// TwinCAT 3 PLC project mdx91test
// ProgramVersion: 3.1.4023.0
// libraries:
//   Tc2_Standard, * (Beckhoff Automation GmbH)
//   Tc2_System, * (Beckhoff Automation GmbH)
//   Tc3_Module, * (Beckhoff Automation GmbH)
// project tree:
//   / PlcTask.TcTTO
//   POUs/ MAIN.TcPOU
//   POUs/SEW_MOVIKITpositioningDrive/ FB_MOVIKITpositioningDrive.TcPOU
//   POUs/SEW_MOVIKITpositioningDrive/General/ eMOVIKITpositioningDrive_ApplMode.TcDUT, stMOVIKITpositioningDrive.TcDUT, stPositioning_IN.TcDUT, stPositioning_OUT.TcDUT
// real-time tasks:
//   TASK PlcTask: cycle T#10ms, priority 20, ADS port 350
// motion (NC):
//   TASK NC-Task 1 SAF: cycle T#2ms, priority 4, ADS port 501
//   TASK NC-Task 1 SVB: cycle T#10ms, priority 8, ADS port 511
//   AXIS Axis 1 (id 1)
//     OtherSettings: AllowMotionCmdToSlave=true
//     encoder EncType=1
//     drive DrvType=5
//       Analog: TorqueSetpointScale=10, ScaleFactorActTorque=0.1
//       TimeComp: TaskDelayCycles=1
//     controller CtrType=1
//       CtrPara: PriorControlFactor=1
//         Observer: BandWidth=20
// I/O:
//   DEVICE Device 5 (EtherCAT), AmsNetId 172.18.214.28.6.1
//     Box 1 (MOVI-C MOVIDRIVE) [MOVI-C MOVIDRIVE]
//       modules: Module 1 (Standard 16 PD)
// variable links:
//   mdx91test/mdx91test Instance <-> Device 5 (EtherCAT)/Box 1 (MOVI-C MOVIDRIVE)
//     PlcTask Inputs/MAIN.stDrive.IN.arrProcessdata_IN <-> Module 1 (Standard 16 PD)/Inputs 16 PD/PI 1
//     PlcTask Inputs/MAIN.stDrive.IN.arrProcessdata_IN @bit {16..112 step 16} <-> Module 1 (Standard 16 PD)/Inputs 16 PD/PI {2..8}  (7 links)
//     PlcTask Outputs/MAIN.stDrive.OUT.arrProcessdata_OUT[{0..7}] <-> Module 1 (Standard 16 PD)/Outputs 16 PD/PO {1..8}  (8 links)

CONFIGURATION mdx91test
    RESOURCE PLC ON TwinCAT3
        TASK PlcTask(INTERVAL := T#10ms, PRIORITY := 20);
        PROGRAM MAIN WITH PlcTask : MAIN;
    END_RESOURCE
END_CONFIGURATION

// ---- POUs/SEW_MOVIKITpositioningDrive/General/eMOVIKITpositioningDrive_ApplMode.TcDUT
{attribute 'qualified_only'}

TYPE eMOVIKITpositioningDrive_ApplMode :
(
	NoModeAssigned := 0,
	JogPosition := 100,
	JogVelocity := 101,
	Velocity := 200,
	ReferenceOffsParam := 300,
	ReferenceOffsFieldb := 301,
	PositionAbs := 400,
	PositionRel := 401,
	PositionModPos := 402,
	PositionModNeg := 403,
	PositionModShort := 404,
	PositionAbsNoRef := 405,
	PositionTouchProbe := 420
)UINT;
END_TYPE

// ---- POUs/SEW_MOVIKITpositioningDrive/General/stMOVIKITpositioningDrive.TcDUT
TYPE stMOVIKITpositioningDrive :
STRUCT
	IN: stPositioning_IN;
	OUT: stPositioning_OUT;
	ApplicationMode: eMOVIKITpositioningDrive_ApplMode;
	
END_STRUCT
END_TYPE

// ---- POUs/SEW_MOVIKITpositioningDrive/General/stPositioning_IN.TcDUT
TYPE stPositioning_IN :
STRUCT
	arrProcessdata_IN AT %I*: ARRAY[0..7] OF UINT;
		
	bEnableEmergencyStop: BOOL;
	bEnableApplicationStop: BOOL;
	bReleaseBrake: BOOL;
	bJogPositive: BOOL;
	bJogNegative: BOOL;
	bApplyRelPos: BOOL;
	bStartStop: BOOL;
	bFaultReset: BOOL;
	bActivateDriveTrain2: BOOL;
	bDeactivateSWLimitSwitch: BOOL;
	bActivateOutputstageInhibit: BOOL;
	bActivateStandBy: BOOL;
	bHAndshakeIN: BOOL;
	bActivateHandShake: BOOL;
		
	iSetpointSpeed: INT;
	uiAcceleration: UINT;
	uiDeceleration: UINT;
	eTargetApplMode: eMOVIKITpositioningDrive_ApplMode;
	diTargetPosition: DINT;
	uiPosMulitplier: UINT;
	
	bDIO01_DO: BOOL;
	bDIO02_DO: BOOL;
	
	

END_STRUCT
END_TYPE

// ---- POUs/SEW_MOVIKITpositioningDrive/General/stPositioning_OUT.TcDUT
TYPE stPositioning_OUT :
STRUCT
	arrProcessdata_OUT AT %Q*: ARRAY[0..7] OF UINT;
	
	bInverterReady: BOOL;
	bSTOinactive: BOOL;
	bOutputstageEnabled: BOOL;
	bBrakeReleased: BOOL;
	bMotorRunning: BOOL;
	bActiveDriveReferenced: BOOL;
	bNewRelPosApplied: BOOL;
	bInPosition: BOOL;
	bFault: BOOL;
	bWarning: BOOL;
	bDriveTrain2Active: BOOL;
	bSpeedComparisonActive:BOOL;
	bSWLimitSwitchInactive: BOOL;
	bStandByModeActive: BOOL;
	bHandshakeOUT: BOOL;
	
	iActualSpeed: INT;
	uiStatus: UINT;
	uiFaultNo: UINT;
	uiWarningNo: UINT;
	uiSubFaultNo: UINT;
	uiActualTorque: UINT;
	
	eActualApplMode: eMOVIKITpositioningDrive_ApplMode;
	diActualPosition: DINT;
	
	
	bDI00: BOOL;
	bDI01: BOOL;
	bDI02: BOOL;
	bDI03: BOOL;
	bDI04: BOOL;
	bDI05: BOOL;
	bDI06: BOOL;
	bDI07: BOOL;
	bDI08: BOOL;
	bDIO01_DI: BOOL;
	bDIO02_DI: BOOL;
	

END_STRUCT
END_TYPE

// ---- POUs/MAIN.TcPOU
PROGRAM MAIN
VAR
	//Axis
	positionDrive: FB_MOVIKITpositioningDrive;
	stDrive: stMOVIKITpositioningDrive;
	
	//Logic
	_uiState			: UINT;
END_VAR

//Beispiel Aufruf mit zentraler Struktur als Referenz übergeben
//positionDrive(example_stMovikitpositioningDrive := positionDriveStruct);

MotorMovementStateMachine();

MapStructureToMovicKitFB();

ACTION MapStructureToMovicKitFB:
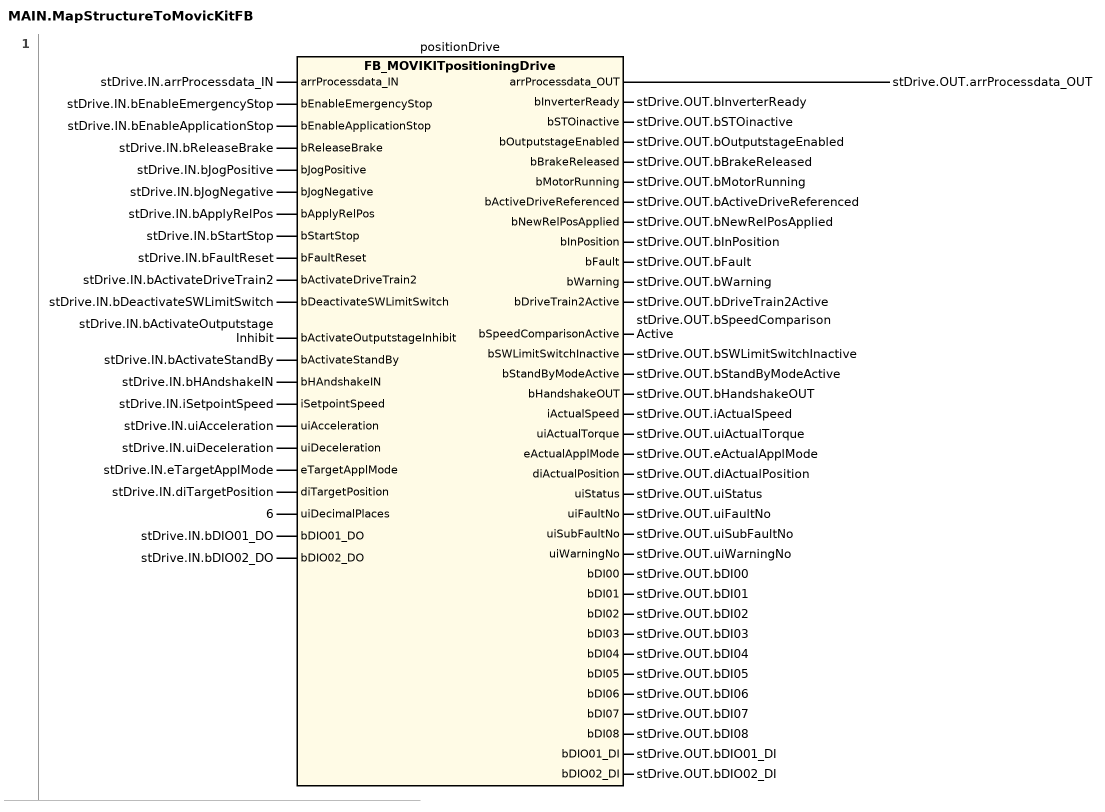
// NETWORK 1
positionDrive(
    arrProcessdata_IN := stDrive.IN.arrProcessdata_IN,
    bEnableEmergencyStop := stDrive.IN.bEnableEmergencyStop,
    bEnableApplicationStop := stDrive.IN.bEnableApplicationStop,
    bReleaseBrake := stDrive.IN.bReleaseBrake,
    bJogPositive := stDrive.IN.bJogPositive,
    bJogNegative := stDrive.IN.bJogNegative,
    bApplyRelPos := stDrive.IN.bApplyRelPos,
    bStartStop := stDrive.IN.bStartStop,
    bFaultReset := stDrive.IN.bFaultReset,
    bActivateDriveTrain2 := stDrive.IN.bActivateDriveTrain2,
    bDeactivateSWLimitSwitch := stDrive.IN.bDeactivateSWLimitSwitch,
    bActivateOutputstageInhibit := stDrive.IN.bActivateOutputstageInhibit,
    bActivateStandBy := stDrive.IN.bActivateStandBy,
    bHAndshakeIN := stDrive.IN.bHAndshakeIN,
    iSetpointSpeed := stDrive.IN.iSetpointSpeed,
    uiAcceleration := stDrive.IN.uiAcceleration,
    uiDeceleration := stDrive.IN.uiDeceleration,
    eTargetApplMode := stDrive.IN.eTargetApplMode,
    diTargetPosition := stDrive.IN.diTargetPosition,
    uiDecimalPlaces := 6,
    bDIO01_DO := stDrive.IN.bDIO01_DO,
    bDIO02_DO := stDrive.IN.bDIO02_DO,
    bInverterReady => stDrive.OUT.bInverterReady,
    bSTOinactive => stDrive.OUT.bSTOinactive,
    bOutputstageEnabled => stDrive.OUT.bOutputstageEnabled,
    bBrakeReleased => stDrive.OUT.bBrakeReleased,
    bMotorRunning => stDrive.OUT.bMotorRunning,
    bActiveDriveReferenced => stDrive.OUT.bActiveDriveReferenced,
    bNewRelPosApplied => stDrive.OUT.bNewRelPosApplied,
    bInPosition => stDrive.OUT.bInPosition,
    bFault => stDrive.OUT.bFault,
    bWarning => stDrive.OUT.bWarning,
    bDriveTrain2Active => stDrive.OUT.bDriveTrain2Active,
    bSpeedComparisonActive => stDrive.OUT.bSpeedComparisonActive,
    bSWLimitSwitchInactive => stDrive.OUT.bSWLimitSwitchInactive,
    bStandByModeActive => stDrive.OUT.bStandByModeActive,
    bHandshakeOUT => stDrive.OUT.bHandshakeOUT,
    iActualSpeed => stDrive.OUT.iActualSpeed,
    uiActualTorque => stDrive.OUT.uiActualTorque,
    eActualApplMode => stDrive.OUT.eActualApplMode,
    diActualPosition => stDrive.OUT.diActualPosition,
    uiStatus => stDrive.OUT.uiStatus,
    uiFaultNo => stDrive.OUT.uiFaultNo,
    uiSubFaultNo => stDrive.OUT.uiSubFaultNo,
    uiWarningNo => stDrive.OUT.uiWarningNo,
    bDI00 => stDrive.OUT.bDI00,
    bDI01 => stDrive.OUT.bDI01,
    bDI02 => stDrive.OUT.bDI02,
    bDI03 => stDrive.OUT.bDI03,
    bDI04 => stDrive.OUT.bDI04,
    bDI05 => stDrive.OUT.bDI05,
    bDI06 => stDrive.OUT.bDI06,
    bDI07 => stDrive.OUT.bDI07,
    bDI08 => stDrive.OUT.bDI08,
    bDIO01_DI => stDrive.OUT.bDIO01_DI,
    bDIO02_DI => stDrive.OUT.bDIO02_DI); // FB_MOVIKITpositioningDrive
stDrive.OUT.arrProcessdata_OUT := positionDrive.arrProcessdata_OUT;
END_ACTION

ACTION MotorMovementStateMachine:
CASE _uiState OF
	
	//Initialisieren
	0:
		IF NOT stDrive.Out.bFault THEN
			_uiState := 10;
		END_IF

	//Generiere Fahrbefehl auf 0mm
	10:
		stDrive.IN.eTargetApplMode			:= eMOVIKITpositioningDrive_ApplMode.PositionAbs;
		stDrive.IN.bEnableApplicationStop	:= TRUE;		//TRUE = Freigabe
		stDrive.IN.bEnableEmergencyStop		:= TRUE;		//TRUE = Freigabe
		stDrive.IN.uiAcceleration			:= 100;			//[Anwendereinheit in der Achse]
		stDrive.IN.uiDeceleration			:= 100;			//[Anwendereinheit in der Achse]
		stDrive.IN.iSetpointSpeed			:= 30;			//[Anwendereinheit in der Achse]
		stDrive.IN.diTargetPosition			:= 0;			//[Anwendereinheit in der Achse]
		stDrive.IN.bStartStop				:= TRUE;		//TRUE = Freigabe Positionierbefehl
		_uiState := 20;
		
		
		
	//Warte auf Achse in Position
	20:
		//Varianten für In pos abfragen
		//1. zeitverzögert fragen
		//2. Istposition abgleichen mit Sollposition
			IF ABS(stDrive.OUT.diActualPosition - stDrive.IN.diTargetPosition) < 1 THEN
				_uiState := 30;
			END_IF
	

	30:
	//Generiere Fahrbefehl auf 1000mm
		stDrive.IN.eTargetApplMode			:= eMOVIKITpositioningDrive_ApplMode.PositionAbs;
		stDrive.IN.bEnableApplicationStop	:= TRUE;		//TRUE = Freigabe
		stDrive.IN.bEnableEmergencyStop		:= TRUE;		//TRUE = Freigabe
		stDrive.IN.uiAcceleration			:= 100;			//[Anwendereinheit in der Achse]
		stDrive.IN.uiDeceleration			:= 100;			//[Anwendereinheit in der Achse]
		stDrive.IN.iSetpointSpeed			:= 30;			//[Anwendereinheit in der Achse]
		stDrive.IN.diTargetPosition			:= 1000;			//[Anwendereinheit in der Achse]
		stDrive.IN.bStartStop				:= TRUE;		//TRUE = Freigabe Positionierbefehl
		_uiState := 35;	

		
	35:
		//Warte auf Achse in Position
		//Varianten für In pos abfragen
		//1. zeitverzögert fragen
		//2. Istposition abgleichen mit Sollposition
			IF ABS(stDrive.OUT.diActualPosition - stDrive.IN.diTargetPosition) < 1 THEN
				_uiState := 10;
			END_IF	
	
	
	//Antrieb stoppen
	40:
		//Variante 1: Antrieb verbleibt in Lageregelung (Motor bestromt)
		stDrive.IN.bStartStop				:= FALSE;		//TRUE = Freigabe Positionierbefehl
		
		//Variante 2: Antrieb lässt Bremse einfallen und beendet Bestromung
		stDrive.IN.bEnableApplicationStop	:= FALSE;		//TRUE = Freigabe

END_CASE
END_ACTION

END_PROGRAM

// ---- POUs/SEW_MOVIKITpositioningDrive/FB_MOVIKITpositioningDrive.TcPOU
FUNCTION_BLOCK FB_MOVIKITpositioningDrive
VAR_INPUT
	//example_stMovikitpositioningDrive : REFERENCE TO stMOVIKITpositioningDrive;	

	arrProcessdata_IN: ARRAY[0..7] OF UINT;
	bEnableEmergencyStop: BOOL;
	bEnableApplicationStop: BOOL;
	bReleaseBrake: BOOL;
	bJogPositive: BOOL;
	bJogNegative: BOOL;
	bApplyRelPos: BOOL;
	bStartStop: BOOL;
	bFaultReset: BOOL;
	bActivateDriveTrain2: BOOL;
	bDeactivateSWLimitSwitch: BOOL;
	bActivateOutputstageInhibit: BOOL;
	bActivateStandBy: BOOL;
	bHAndshakeIN: BOOL;
	
		
	iSetpointSpeed: INT;
	uiAcceleration: UINT;
	uiDeceleration: UINT;
	eTargetApplMode: eMOVIKITpositioningDrive_ApplMode;
	diTargetPosition: DINT;
	uiDecimalPlaces: UINT;
	
	bDIO01_DO: BOOL;
	bDIO02_DO: BOOL;
	
	
END_VAR
VAR_OUTPUT
	arrProcessdata_OUT: ARRAY[0..7] OF UINT;
	bInverterReady: BOOL;
	bSTOinactive: BOOL;
	bOutputstageEnabled: BOOL;
	bBrakeReleased: BOOL;
	bMotorRunning: BOOL;
	bActiveDriveReferenced: BOOL;
	bNewRelPosApplied: BOOL;
	bInPosition: BOOL;
	bFault: BOOL;
	bWarning: BOOL;
	bDriveTrain2Active: BOOL;
	bSpeedComparisonActive:BOOL;
	bSWLimitSwitchInactive: BOOL;
	bStandByModeActive: BOOL;
	bHandshakeOUT: BOOL;
	
	iActualSpeed: INT;
	uiActualTorque: UINT;
	eActualApplMode: eMOVIKITpositioningDrive_ApplMode;
	diActualPosition: DINT;
	
	uiStatus: UINT;
	uiFaultNo: UINT;
	uiSubFaultNo: UINT;
	uiWarningNo: UINT;
	
	
	
	
	bDI00: BOOL;
	bDI01: BOOL;
	bDI02: BOOL;
	bDI03: BOOL;
	bDI04: BOOL;
	bDI05: BOOL;
	bDI06: BOOL;
	bDI07: BOOL;
	bDI08: BOOL;
	bDIO01_DI: BOOL;
	bDIO02_DI: BOOL;
END_VAR
VAR
	uiFaultStatus_i: UINT;
	uiSetPosHigh_i: UINT;
	uiSetPosLow_i: UINT;
	uiActPosHigh_i: DINT;
	uiActPosLow_i: DINT;
	uiStatus_SubFault_i: UINT;
	uiActualApplMode_i: UINT;
END_VAR

//================================================================================================================
//
//	This Beckhoff TwinCAT 3 function block is a sample program for controlling the drive using 
//	"MOVIKITdrive positioning" via fieldbus on MOVI-C(R) inverters.
//	It is an open function block and may be changed by the customer to his needs.
//	
//	Liability/Disclaimer
//	--------------------
//	This sample program outlines a basic approach for informational and demonstration purposes only. 
//	The User understands and agrees that SEW-EURODRIVE has made no representation or warranty hereunder, 
//	expressed or implied, as to the accuracy or completeness of the sample program software, 
//	and shall have NO liability hereunder to the User or its Representatives relating to or resulting 
//	from the use of the sample program software or any errors therein or omissions therefrom.
//
//	Change Log
//	----------
//	- Creation Date: 	2021-04-14	
//	- V1.0				2021-04-14	
//
//	co-applicable software
//	----------------------
//	For using the function block the following STRUCS and ENUMS may also be imported
//	- eMOVIKITpositioningDrive_ApplMode 	(ENUM)
//	- stMOVIKITpositioningDrive				(STRUCT)
//	- stPositioning_IN						(STRUCT)
//	- stPositioning_OUT						(STRUCT)
//
//==================================================================================================================


IF uiDecimalPlaces=0 THEN
	uiDecimalPlaces := 1;
END_IF

diTargetPosition := diTargetPosition*uiDecimalPlaces;
uiSetPosLow_i := DINT_TO_UINT(diTargetPosition AND 16#0000FFFF); 
uiSetPosHigh_i := DINT_TO_UINT(SHR(diTargetPosition,16)); 

(*====================================================================================
	Control --> PO
=====================================================================================*)
arrProcessdata_OUT[0].0 := bEnableEmergencyStop;
arrProcessdata_OUT[0].1 := bEnableApplicationStop;
arrProcessdata_OUT[0].3 := bReleaseBrake;
arrProcessdata_OUT[0].4 := bJogPositive;
arrProcessdata_OUT[0].5 := bJogNegative;
arrProcessdata_OUT[0].6 := bApplyRelPos;
arrProcessdata_OUT[0].7 := bStartStop;
arrProcessdata_OUT[0].8 := bFaultReset;

arrProcessdata_OUT[0].10 := bActivateDriveTrain2;
arrProcessdata_OUT[0].12 := bDeactivateSWLimitSwitch;
arrProcessdata_OUT[0].13 := bActivateOutputstageInhibit;
arrProcessdata_OUT[0].14 := bActivateStandBy;
arrProcessdata_OUT[0].15 := bHAndshakeIN;


arrProcessdata_OUT[1] := iSetpointSpeed;
arrProcessdata_OUT[2] := uiAcceleration;
arrProcessdata_OUT[3] := uiDeceleration;

arrProcessdata_OUT[4].0 := bDIO01_DO;
arrProcessdata_OUT[4].1 := bDIO02_DO;

arrProcessdata_OUT[5] := eTargetApplMode;

arrProcessdata_OUT[6] := uiSetPosHigh_i;
arrProcessdata_OUT[7] := uiSetPosLow_i;

(*====================================================================================
	PI --> Status
=====================================================================================*)
bInverterReady := arrProcessdata_IN[0].0;
bSTOinactive := arrProcessdata_IN[0].1;
bOutputstageEnabled := arrProcessdata_IN[0].2;
bBrakeReleased := arrProcessdata_IN[0].3;
bMotorRunning := arrProcessdata_IN[0].4;
bActiveDriveReferenced := arrProcessdata_IN[0].5;
bNewRelPosApplied := arrProcessdata_IN[0].6;
bInPosition := arrProcessdata_IN[0].7;
bFault := arrProcessdata_IN[0].8;
bWarning := arrProcessdata_IN[0].9;
bDriveTrain2Active := arrProcessdata_IN[0].10;
bSpeedComparisonActive := arrProcessdata_IN[0].11;
bSWLimitSwitchInactive := arrProcessdata_IN[0].12;
bStandByModeActive := arrProcessdata_IN[0].14;
bHandshakeOUT := arrProcessdata_IN[0].15;

iActualSpeed:= arrProcessdata_IN[1];
uiStatus_SubFault_i := arrProcessdata_IN[2] AND 16#0F; 
uiFaultStatus_i := SHR(arrProcessdata_IN[2],8);




IF NOT bFault AND NOT bWarning THEN
	uiStatus := uiStatus_SubFault_i;
	uiFaultNo := 0;
	uiSubFaultNo := 0;
	uiWarningNo := 0;
ELSE
	uiStatus := 0;
	
	IF bWarning THEN
		uiFaultNo := 0;
		uiSubFaultNo := 0;
		uiWarningNo := uiFaultStatus_i;
	ELSIF bFault THEN
		uiFaultNo := uiFaultStatus_i;
		uiSubFaultNo := uiStatus_SubFault_i;
		uiWarningNo := 0;
	END_IF
		
END_IF

uiActualTorque:= arrProcessdata_IN[3];

bDI00 := arrProcessdata_IN[4].0;
bDI01 := arrProcessdata_IN[4].1;
bDI02 := arrProcessdata_IN[4].2;
bDI03 := arrProcessdata_IN[4].3;
bDI04 := arrProcessdata_IN[4].4;
bDI05 := arrProcessdata_IN[4].5;
bDI06 := arrProcessdata_IN[4].6;
bDI07 := arrProcessdata_IN[4].7;
bDI08 := arrProcessdata_IN[4].8;

eActualApplMode := arrProcessdata_IN[5];


uiActPosLow_i := UINT_TO_DWORD(arrProcessdata_IN[7]);
uiActPosHigh_i := SHL(UINT_TO_DWORD(arrProcessdata_IN[6]),16);
diActualPosition := (uiActPosHigh_i + uiActPosLow_i)/uiDecimalPlaces;

END_FUNCTION_BLOCK
